FUNCTION_BLOCK AI_SUBSCRIBE_1 (* Subscribe to a PUBLISH_1 Block and buffer the received INT with a D_FF *)
  (* Standard: 61499-2; Description: Copyright (c) 2026 HR Agrartechnik GmbH This program and the accompanying materials are made available under the terms of the Eclipse Public License 2.0 which is available at https://www.eclipse.org/legal/epl-2.0/ SPDX-License-Identifier: EPL-2.0 *)
  (* Version 1.0, 2026-08-07, Franz Höpfinger, HR Agrartechnik GmbH, initial API and implementation and/or initial documentation *)
  PACKAGE adapter::net;
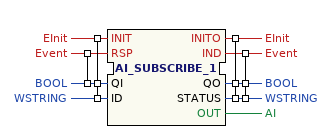
  EVENT_INPUT
    INIT : EInit WITH QI, ID; (* Initialization *)
    RSP WITH QI; (* Response to the received data *)
  END_EVENT
  EVENT_OUTPUT
    INITO : EInit WITH QO, STATUS; (* Initialization Confirm *)
    IND WITH QO, STATUS; (* New data available *)
  END_EVENT
  VAR_INPUT
    QI : BOOL;
    ID : WSTRING;
  END_VAR
  VAR_OUTPUT
    QO : BOOL;
    STATUS : WSTRING;
  END_VAR
  PLUGS
    OUT : adapter::types::unidirectional::AI; (* Buffered received INT *)
  END_PLUGS
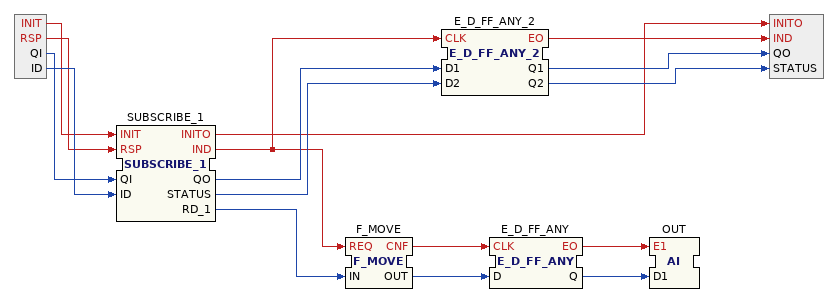
  FBS
    SUBSCRIBE_1 : iec61499::net::SUBSCRIBE_1;
    E_D_FF_ANY : iec61499::events::E_D_FF_ANY;
    F_MOVE : iec61131::selection::F_MOVE; {SET_ATTRIBUTE(DataType, INT)}
    E_D_FF_ANY_2 : iec61499::events::E_D_FF_ANY_2;
  END_FBS
  EVENT_CONNECTIONS
    INIT TO SUBSCRIBE_1.INIT;
    RSP TO SUBSCRIBE_1.RSP;
    SUBSCRIBE_1.INITO TO INITO;
    SUBSCRIBE_1.IND TO F_MOVE.REQ;
    E_D_FF_ANY.EO TO OUT.E1;
    F_MOVE.CNF TO E_D_FF_ANY.CLK;
    SUBSCRIBE_1.IND TO E_D_FF_ANY_2.CLK;
    E_D_FF_ANY_2.EO TO IND;
  END_CONNECTIONS
  DATA_CONNECTIONS
    QI TO SUBSCRIBE_1.QI;
    ID TO SUBSCRIBE_1.ID;
    SUBSCRIBE_1.QO TO E_D_FF_ANY_2.D1;
    SUBSCRIBE_1.STATUS TO E_D_FF_ANY_2.D2;
    SUBSCRIBE_1.RD_1 TO F_MOVE.IN;
    E_D_FF_ANY.Q TO OUT.D1;
    F_MOVE.OUT TO E_D_FF_ANY.D;
    E_D_FF_ANY_2.Q1 TO QO;
    E_D_FF_ANY_2.Q2 TO STATUS;
  END_CONNECTIONS
END_FUNCTION_BLOCK
